FUNCTION_BLOCK CLIENT_1 (* Connect to a SERVER_1 Block *)
  (* Standard: 61499-2; Description: Copyright (c) 2017 fortiss GmbH This program and the accompanying materials are made available under the terms of the Eclipse Public License 2.0 which is available at https://www.eclipse.org/legal/epl-2.0/ SPDX-License-Identifier: EPL-2.0 *)
  (* Version 1.0, 2017-10-25, Alois Zoitl, fortiss GmbH, initial API and implementation and/or initial documentation *)
  (* Version 3.0, 2025-04-14, Patrick Aigner, changed package *)
  PACKAGE iec61499::net;
  {SET_ATTRIBUTE(eclipse4diac::core::GenericClassName, 'GEN_CLIENT')}
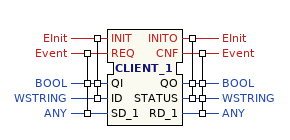
  EVENT_INPUT
    INIT : EInit WITH QI, ID; (* Open new connection (QI = TRUE) / Close connection (QI = FALSE) *)
    REQ WITH QI, SD_1; (* Send data to Server, Request Data from Server *)
  END_EVENT
  EVENT_OUTPUT
    INITO : EInit WITH QO, STATUS; (* New connection established (QI = TRUE) / connection closed (QI = FALSE) *)
    CNF WITH QO, STATUS, RD_1; (* New data available from Server *)
  END_EVENT
  VAR_INPUT
    QI : BOOL;
    ID : WSTRING;
    SD_1 : ANY;
  END_VAR
  VAR_OUTPUT
    QO : BOOL;
    STATUS : WSTRING;
    RD_1 : ANY;
  END_VAR
END_FUNCTION_BLOCK
